KUKA KRL data list: hmi.dat

&ACCESS RVO
&REL 6
&PARAM EDITMASK = *
&PARAM TEMPLATE = C:\KRC\Roboter\Template\ExpertVorgabe
DEFDAT hmi PUBLIC

ENDDAT
